FUNCTION_BLOCK StartStopSpPv (* Basic Function Block Type *)
  (* Standard: 61499-2 *)
  (* Version 0.0, 7/21/2026, Schneider Electric, Template *)
  PACKAGE SE.Nereda;
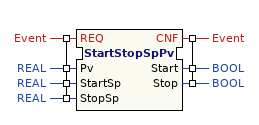
  EVENT_INPUT
    REQ WITH Pv, StartSp, StopSp; (* Normal Execution Request *)
  END_EVENT
  EVENT_OUTPUT
    CNF WITH Start, Stop; (* Execution Confirmation *)
  END_EVENT
  VAR_INPUT
    Pv : REAL;
    StartSp : REAL;
    StopSp : REAL;
  END_VAR
  VAR_OUTPUT
    Start : BOOL;
    Stop : BOOL;
  END_VAR
  VAR
    FirstStart : BOOL := FALSE;
  END_VAR
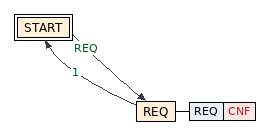
  EC_STATES
    START; (* Initial State *)
    REQ : REQ -> CNF; (* Normal execution *)
  END_STATES
  EC_TRANSITIONS
    START TO REQ := REQ;
    REQ TO START := 1;
  END_TRANSITIONS
  ALGORITHM REQ IN ST: (* Normally executed algorithm *)
;
IF Pv >= StartSp THEN
	FirstStart := TRUE;
	Start := TRUE;
	Stop := FALSE;
END_IF;

IF Pv <= StopSp OR NOT FirstStart THEN
	Start := FALSE;
	Stop := TRUE;
END_IF;
  END_ALGORITHM
END_FUNCTION_BLOCK
